FUNCTION_BLOCK SS5_ifb_ps_Raiser_n_Flipper (* Composite FB wrapping other FBs *)
  (* Standard: 61499-2 *)
  (* Version 1.0, 2025-07-23, PS_Transformer_for_Unknown *)
  PACKAGE UserLibs::SubStations::SS5;
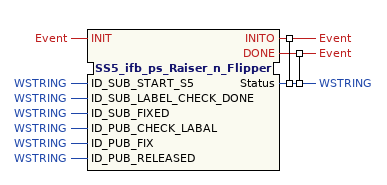
  EVENT_INPUT
    INIT; (* Initialization Request *)
  END_EVENT
  EVENT_OUTPUT
    INITO WITH Status; (* Initialization Confirm *)
    DONE WITH Status; (* Execution Confirmation *)
  END_EVENT
  VAR_INPUT
    ID_SUB_START_S5 : WSTRING;
    ID_SUB_LABEL_CHECK_DONE : WSTRING;
    ID_SUB_FIXED : WSTRING;
    ID_PUB_CHECK_LABAL : WSTRING;
    ID_PUB_FIX : WSTRING;
    ID_PUB_RELEASED : WSTRING;
  END_VAR
  VAR_OUTPUT
    Status : WSTRING; (* Output event qualifier *)
  END_VAR
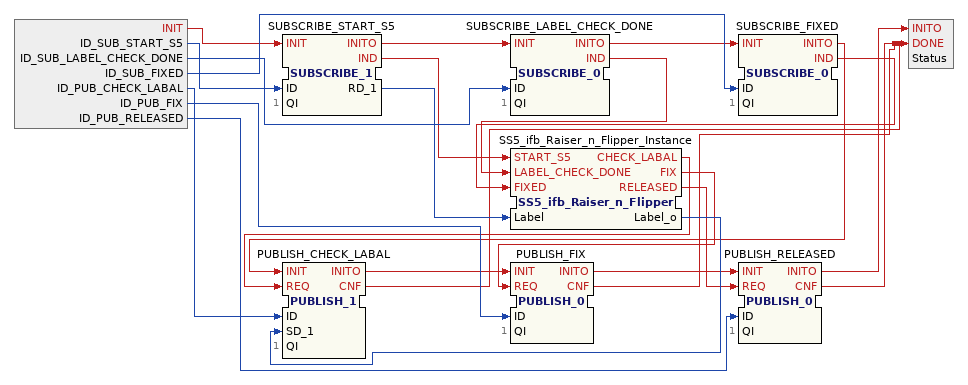
  FBS
    SS5_ifb_Raiser_n_Flipper_Instance : SS5_ifb_Raiser_n_Flipper;
    SUBSCRIBE_START_S5 : SUBSCRIBE_1(QI := 1);
    SUBSCRIBE_LABEL_CHECK_DONE : SUBSCRIBE_0(QI := 1);
    SUBSCRIBE_FIXED : SUBSCRIBE_0(QI := 1);
    PUBLISH_CHECK_LABAL : PUBLISH_1(QI := 1);
    PUBLISH_FIX : PUBLISH_0(QI := 1);
    PUBLISH_RELEASED : PUBLISH_0(QI := 1);
  END_FBS
  EVENT_CONNECTIONS
    INIT TO SUBSCRIBE_START_S5.INIT;
    SUBSCRIBE_START_S5.INITO TO SUBSCRIBE_LABEL_CHECK_DONE.INIT;
    SUBSCRIBE_LABEL_CHECK_DONE.INITO TO SUBSCRIBE_FIXED.INIT;
    SUBSCRIBE_FIXED.INITO TO PUBLISH_CHECK_LABAL.INIT;
    PUBLISH_CHECK_LABAL.INITO TO PUBLISH_FIX.INIT;
    PUBLISH_FIX.INITO TO PUBLISH_RELEASED.INIT;
    PUBLISH_RELEASED.INITO TO INITO;
    SUBSCRIBE_START_S5.IND TO SS5_ifb_Raiser_n_Flipper_Instance.START_S5;
    SUBSCRIBE_LABEL_CHECK_DONE.IND TO SS5_ifb_Raiser_n_Flipper_Instance.LABEL_CHECK_DONE;
    SUBSCRIBE_FIXED.IND TO SS5_ifb_Raiser_n_Flipper_Instance.FIXED;
    SS5_ifb_Raiser_n_Flipper_Instance.CHECK_LABAL TO PUBLISH_CHECK_LABAL.REQ;
    SS5_ifb_Raiser_n_Flipper_Instance.FIX TO PUBLISH_FIX.REQ;
    SS5_ifb_Raiser_n_Flipper_Instance.RELEASED TO PUBLISH_RELEASED.REQ;
    PUBLISH_CHECK_LABAL.CNF TO DONE;
    PUBLISH_FIX.CNF TO DONE;
    PUBLISH_RELEASED.CNF TO DONE;
  END_CONNECTIONS
  DATA_CONNECTIONS
    ID_SUB_START_S5 TO SUBSCRIBE_START_S5.ID;
    ID_SUB_LABEL_CHECK_DONE TO SUBSCRIBE_LABEL_CHECK_DONE.ID;
    ID_SUB_FIXED TO SUBSCRIBE_FIXED.ID;
    ID_PUB_CHECK_LABAL TO PUBLISH_CHECK_LABAL.ID;
    ID_PUB_FIX TO PUBLISH_FIX.ID;
    ID_PUB_RELEASED TO PUBLISH_RELEASED.ID;
    SUBSCRIBE_START_S5.RD_1 TO SS5_ifb_Raiser_n_Flipper_Instance.Label;
    SS5_ifb_Raiser_n_Flipper_Instance.Label_o TO PUBLISH_CHECK_LABAL.SD_1;
  END_CONNECTIONS
END_FUNCTION_BLOCK
